// TIA Portal project "FactoryIO_Template_S7-1200_V16_V16" (V16)
// Vorlageprojekt für das Buch mit Zielsystem S7-1200

(* hardware
DEVICE "S7-1200-Station_1"  S7-1200 Station
   slot 0: "Baugruppenträger_0"  Rack  V1.0
   slot 1: "PLC_1"  CPU 1211C DC/DC/DC  6ES7 211-1AE40-0XB0  V4.1
*)

// ===== PLC "PLC_1"  CPU 1211C DC/DC/DC =====

VAR_GLOBAL   // PLC tag table "Standard-Variablentabelle"
   "2F conveyor" AT %A0.0 : Bool;
   "start" AT %E0.0 : Bool;
   "stop" AT %E0.1 : Bool;
   "Tag_4" AT %I10.0 : Bool;
   "Tag_5" AT %Q10.0 : Bool;
   "Tag_6" AT %I10.1 : Bool;
   "TT-back limit" AT %I0.2 : Bool;
   "TT-front limit" AT %I0.3 : Bool;
   "difuse sensor1" AT %I0.4 : Bool;
   "difuse sensor3" AT %I0.5 : Bool;
   "difuse sensor4" AT %I0.6 : Bool;
   "limit 0" AT %I0.7 : Bool;
   "limit 90" AT %I1.0 : Bool;
   "2R conveyor" AT %Q0.1 : Bool;
   "2L conveyor" AT %Q0.2 : Bool;
   "TT Roll +" AT %Q0.3 : Bool;
   "TT Turn" AT %Q0.4 : Bool;
   "TT Roll -" AT %Q0.5 : Bool;
   "loop marker" AT %M0.0 : Bool;
   "dif-sens1-marker" AT %M0.1 : Bool;
   "dif-sens2-marker" AT %M0.2 : Bool;
   "Tag_3" AT %M1.0 : Bool;
   "Tag_7" AT %M1.1 : Bool;
   "turn R-ss" AT %M0.7 : Bool;
   "turn L-ss" AT %M0.6 : Bool;
   "roll+state1" AT %M2.0 : Bool;
   "roll+state2" AT %M2.1 : Bool;
   "Tag_1" AT %M1.2 : Bool;
   "Tag_2" AT %M0.4 : Bool;
END_VAR

FUNCTION "MHJ-PLC-Lab-Function-S71200" : Void   // FC9000, SCL
{ S7_Optimized_Access := 'TRUE' }
VERSION : 0.1
   VAR_TEMP
      rdTimeReturn : Int;
      outputTime : DTL;
      SyncVal : Byte;
      forVal : Int;
      forVal_2 : Int;
      Value : Byte;
   END_VAR
   VAR CONSTANT
      CompVal : Byte := 16#34;
      Value_01 : Byte := 16#11;
      Value_01_DW : DWord := 16#A165_D992;
      Value_02_DW : DWord := 16#58BE_4401;
   END_VAR
BEGIN

   #Value:=PEEK(area := 16#82,
        dbNumber := 0,
        byteOffset := 511);
   #Value := #Value + 1;

   POKE(area := 16#82,
        dbNumber := 0,
        byteOffset := 511,
        value := #Value);

   POKE(area:=16#81,
        dbNumber:=0,
        byteOffset:=1016,
        value:=#Value_01_DW);
   POKE(area := 16#81,
        dbNumber := 0,
        byteOffset := 1020,
        value := #Value_02_DW);

   POKE(area := 16#81,
        dbNumber := 0,
        byteOffset := 511,
        value := B#16#00);

   FOR #forVal := 0 TO 120 DO
       FOR #forVal_2:=0 TO 10 DO
           #rdTimeReturn:=RD_SYS_T(#outputTime);
           #rdTimeReturn := WR_SYS_T(#outputTime);
           #rdTimeReturn := RD_SYS_T(#outputTime);
           #rdTimeReturn := WR_SYS_T(#outputTime);
       END_FOR;
       #SyncVal:= PEEK(area := 16#81,
                      dbNumber := 0,
                      byteOffset := 511);
       IF #SyncVal = #CompVal THEN
          GOTO M_1;
       END_IF;
   END_FOR;
   RETURN;

   M_1:
   POKE(area := 16#81,
        dbNumber := 0,
        byteOffset := 511,
        value := B#16#0);
END_FUNCTION

ORGANIZATION_BLOCK "Main"   // OB1, LAD, ProgramCycle
TITLE = "Main Program Sweep (Cycle)"
{ S7_Optimized_Access := 'TRUE' }
VERSION : 0.1
   VAR_INPUT
      Initial_Call : Bool;   // Initial call of this OB
      Remanence : Bool;   // =True, if remanent data are available
   END_VAR
   VAR_TEMP   // added for the SCL form of the ladder/FBD networks
      _w1 : Bool;
   END_VAR
BEGIN

REGION Network 1: Konnektierungsbaustein für PLC-Lab
   // Im Netzwerk 1 wird der Konnektierungsbaustein für PLC-Lab aufgerufen.
   // Dieser Aufruf darf nicht entfernt werden!
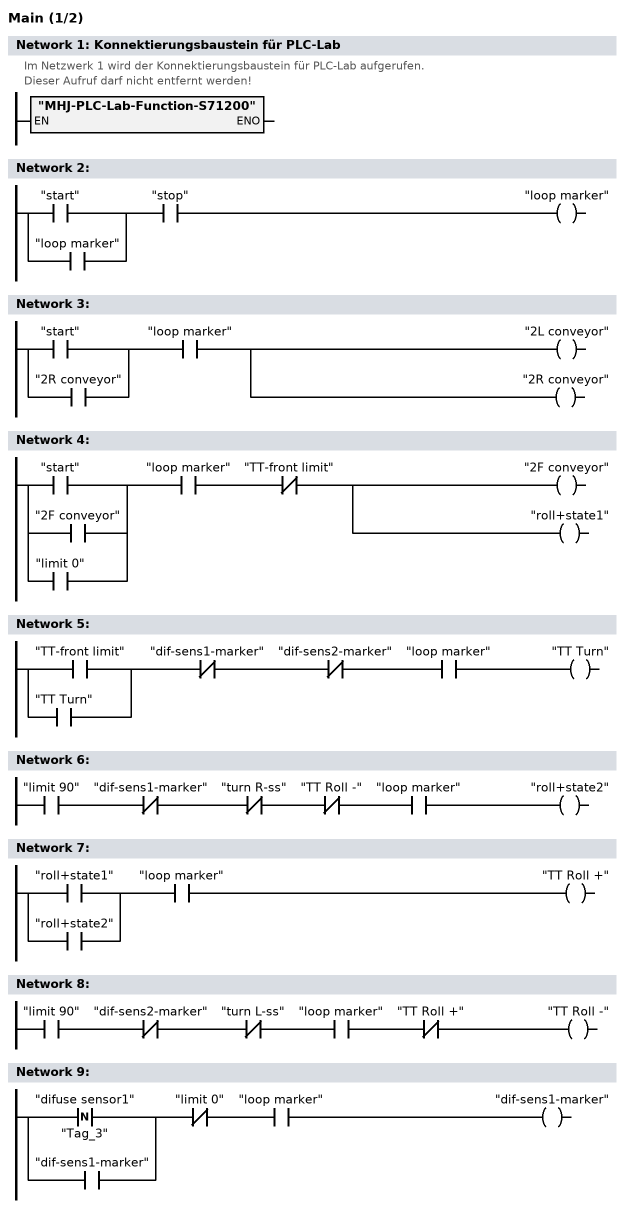
   RUNG wire#powerrail
      "MHJ-PLC-Lab-Function-S71200"()
   END_RUNG
   // the same network as SCL:
   "MHJ-PLC-Lab-Function-S71200"();
END_REGION

REGION Network 2
   RUNG wire#powerrail
      Contact( "start" )
      wire#w1
      Contact( "stop" )
      Coil( "loop marker" )
   END_RUNG
   RUNG wire#powerrail
      Contact( "loop marker" )
   END_RUNG wire#w1
   // the same network as SCL:
   "loop marker" := ("start" OR "loop marker") AND "stop";
END_REGION

REGION Network 3
   RUNG wire#powerrail
      Contact( "start" )
      wire#w1
      Contact( "loop marker" )
      wire#w2
      Coil( "2L conveyor" )
   END_RUNG
   RUNG wire#powerrail
      Contact( "2R conveyor" )
   END_RUNG wire#w1
   RUNG wire#w2
      Coil( "2R conveyor" )
   END_RUNG
   // the same network as SCL:
   "2L conveyor" := ("start" OR "2R conveyor") AND "loop marker";
   "2R conveyor" := "2L conveyor";
END_REGION

REGION Network 4
   RUNG wire#powerrail
      Contact( "start" )
      wire#w1
      Contact( "loop marker" )
      I_Contact( "TT-front limit" )
      wire#w2
      Coil( "2F conveyor" )
   END_RUNG
   RUNG wire#powerrail
      Contact( "2F conveyor" )
   END_RUNG wire#w1
   RUNG wire#powerrail
      Contact( "limit 0" )
   END_RUNG wire#w1
   RUNG wire#w2
      Coil( "roll+state1" )
   END_RUNG
   // the same network as SCL:
   "2F conveyor" := ("start" OR "2F conveyor" OR "limit 0") AND "loop marker" AND NOT "TT-front limit";
   "roll+state1" := "2F conveyor";
END_REGION

REGION Network 5
   RUNG wire#powerrail
      Contact( "TT-front limit" )
      wire#w1
      I_Contact( "dif-sens1-marker" )
      I_Contact( "dif-sens2-marker" )
      Contact( "loop marker" )
      Coil( "TT Turn" )
   END_RUNG
   RUNG wire#powerrail
      Contact( "TT Turn" )
   END_RUNG wire#w1
   // the same network as SCL:
   "TT Turn" := ("TT-front limit" OR "TT Turn") AND NOT "dif-sens1-marker" AND NOT "dif-sens2-marker" AND "loop marker";
END_REGION

REGION Network 6
   RUNG wire#powerrail
      Contact( "limit 90" )
      I_Contact( "dif-sens1-marker" )
      I_Contact( "turn R-ss" )
      I_Contact( "TT Roll -" )
      Contact( "loop marker" )
      Coil( "roll+state2" )
   END_RUNG
   // the same network as SCL:
   "roll+state2" := "limit 90" AND NOT "dif-sens1-marker" AND NOT "turn R-ss" AND NOT "TT Roll -" AND "loop marker";
END_REGION

REGION Network 7
   RUNG wire#powerrail
      Contact( "roll+state1" )
      wire#w1
      Contact( "loop marker" )
      Coil( "TT Roll +" )
   END_RUNG
   RUNG wire#powerrail
      Contact( "roll+state2" )
   END_RUNG wire#w1
   // the same network as SCL:
   "TT Roll +" := ("roll+state1" OR "roll+state2") AND "loop marker";
END_REGION

REGION Network 8
   RUNG wire#powerrail
      Contact( "limit 90" )
      I_Contact( "dif-sens2-marker" )
      I_Contact( "turn L-ss" )
      Contact( "loop marker" )
      I_Contact( "TT Roll +" )
      Coil( "TT Roll -" )
   END_RUNG
   // the same network as SCL:
   "TT Roll -" := "limit 90" AND NOT "dif-sens2-marker" AND NOT "turn L-ss" AND "loop marker" AND NOT "TT Roll +";
END_REGION

REGION Network 9
   RUNG wire#powerrail
      N_Contact(operand := "difuse sensor1", bit := "Tag_3")
      wire#w1
      I_Contact( "limit 0" )
      Contact( "loop marker" )
      Coil( "dif-sens1-marker" )
   END_RUNG
   RUNG wire#powerrail
      Contact( "dif-sens1-marker" )
   END_RUNG wire#w1
   // the same network as SCL:
   #_w1 := NOT "difuse sensor1" AND "Tag_3";   // falling edge of "difuse sensor1"
   "Tag_3" := "difuse sensor1";
   "dif-sens1-marker" := (#_w1 OR "dif-sens1-marker") AND NOT "limit 0" AND "loop marker";
END_REGION

REGION Network 10
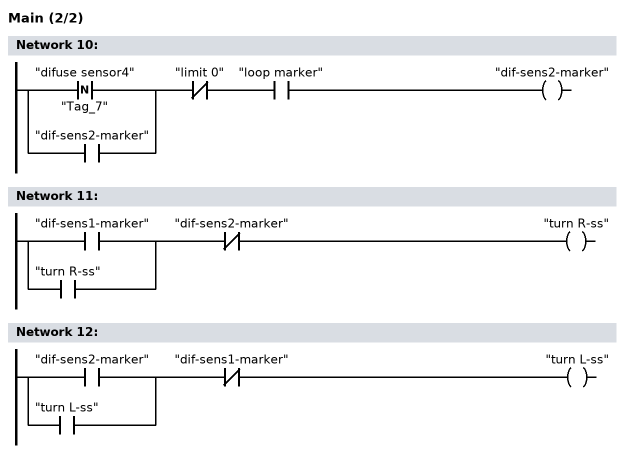
   RUNG wire#powerrail
      N_Contact(operand := "difuse sensor4", bit := "Tag_7")
      wire#w1
      I_Contact( "limit 0" )
      Contact( "loop marker" )
      Coil( "dif-sens2-marker" )
   END_RUNG
   RUNG wire#powerrail
      Contact( "dif-sens2-marker" )
   END_RUNG wire#w1
   // the same network as SCL:
   #_w1 := NOT "difuse sensor4" AND "Tag_7";   // falling edge of "difuse sensor4"
   "Tag_7" := "difuse sensor4";
   "dif-sens2-marker" := (#_w1 OR "dif-sens2-marker") AND NOT "limit 0" AND "loop marker";
END_REGION

REGION Network 11
   RUNG wire#powerrail
      Contact( "dif-sens1-marker" )
      wire#w1
      I_Contact( "dif-sens2-marker" )
      Coil( "turn R-ss" )
   END_RUNG
   RUNG wire#powerrail
      Contact( "turn R-ss" )
   END_RUNG wire#w1
   // the same network as SCL:
   "turn R-ss" := ("dif-sens1-marker" OR "turn R-ss") AND NOT "dif-sens2-marker";
END_REGION

REGION Network 12
   RUNG wire#powerrail
      Contact( "dif-sens2-marker" )
      wire#w1
      I_Contact( "dif-sens1-marker" )
      Coil( "turn L-ss" )
   END_RUNG
   RUNG wire#powerrail
      Contact( "turn L-ss" )
   END_RUNG wire#w1
   // the same network as SCL:
   "turn L-ss" := ("dif-sens2-marker" OR "turn L-ss") AND NOT "dif-sens1-marker";
END_REGION
END_ORGANIZATION_BLOCK